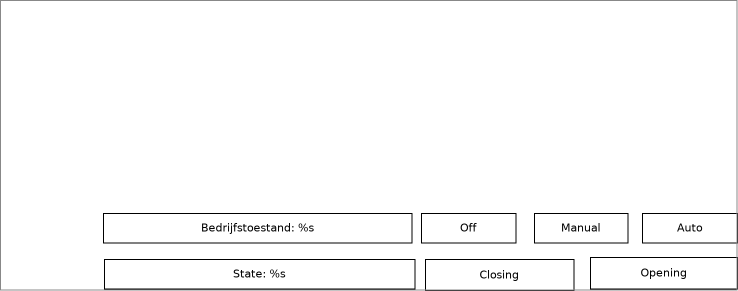
VISUALIZATION Visualization_1  // 738x291
    RoundedRectangle (534,213 94x30), "Manual"
        OnMouseDown: execute { MAIN.V2013_DG.CurrentMode := E_Bedrijfstoestand.manual; }
    RoundedRectangle (421,213 95x30), "Off"
        OnMouseDown: execute { MAIN.V2013_DG.CurrentMode := E_Bedrijfstoestand.off; }
    RoundedRectangle (642,213 96x30), "Auto"
        OnMouseDown: execute { MAIN.V2013_DG.CurrentMode := E_Bedrijfstoestand.auto; }
    RoundedRectangle (103,213 309x30), "Bedrijfstoestand: %s", text variable: MAIN.V2013_DG.currentMode
    RoundedRectangle (104,259 311x30), "State: %s", text variable: MAIN.V2013_DG.currentState
    RoundedRectangle (425,259 149x32), "Closing", colour toggle: MAIN.OutOpeningV2013.internalState
    RoundedRectangle (590,257 148x32), "Opening", colour toggle: MAIN.OutOpeningV2022.internalState
END_VISUALIZATION

(* stored: Version 1.1.0.1, ProductVersion 3.1.4026.8
   Visu Visualization_1: Id {ee736e15-87a1-42c8-9ca9-4369a238693b} *)
